      U     "MAL1S017Par".Ilo.GrCMDManStop[1];
      R     "MAL1S017Par".Ilo.GrCMDManStop[1];
// man fault reset
      U     "MAL1S017Par".Ilo.GrCMDManFaultReset[1];
      S     "G005G".Gr.CmdFaultReset; // GENERAL ELEMENTS GERM 1
      S     "G100M".Gr.CmdFaultReset; // Traveling  Drive Germatingbox 1
      S     "G104M".Gr.CmdFaultReset; // Turning Screws Germinationbox 1
      R     "MAL1S017Par".Ilo.GrCMDManFaultReset[1];
      NOP   0;
// Manual wall locking
      UN    "G099M".Gr.InManual; // Wall locking Germatingbox 1
      ON    "G102M".A_2115_KCL01I5.InpTrue; // pushbutton "locking"
      SPB   f102;
      S     "G099M".Gr.CmdOn; // Wall locking/unlocking Germatingbox 1
f102: NOP   0;
// Manual wall unlocking
      UN    "G099M".Gr.InManual; // Wall locking Germatingbox 1
      ON    "G102M".A_2115_KCL01I6.InpTrue; // pushbutton "unlocking"
      SPB   f103;
      S     "G099M".Gr.CmdOn; // Wall locking/unlocking Germatingbox 1
f103: NOP   0;
// Manual discharger coupling
      UN    "G098M".Gr.InManual; // discharger coupling Germatingbox 1
      ON    "G102M".A_2115_KCL01I4.InpTrue; // pushbutton "discharger coupling"
      SPB   f104;
      S     "G098M".Gr.CmdOn; // discharger coupling Germatingbox 1
f104: NOP   0;
// Manual discharger uncoupling
      UN    "G098M".Gr.InManual; // discharger coupling Germatingbox 1
      ON    "G102M".A_2115_KCL01I3.InpTrue; // pushbutton "discharger uncoupling"
      SPB   f105;
      S     "G098M".Gr.CmdOn; // discharger coupling Germatingbox 1
f105: NOP   0;
// Manual backwall moving
      UN    "G097M".Gr.InManual; // Backwall moving Germatingbox 1
      ON    "G102M".A_2115_KCL01I1.InpTrue; // pushbutton "backwall lifting"
      SPB   f106;
      S     "G097M".Gr.CmdOn; // Backwall moving Germatingbox 1
f106: NOP   0;
      UN    "G097M".Gr.InManual; // Backwall moving Germatingbox 1
      ON    "G102M".A_2115_KCL01I2.InpTrue; // pushbutton "backwall lowerring"
      SPB   f107;
      S     "G097M".Gr.CmdOn; // Backwall moving Germatingbox 1
f107: NOP   0;
// manual direction
      UN    "G100M".Gr.InManual; // Traveling  Drive Germatingbox 1
      O     ;
      UN    "G102M".A_2111_KCL01I3.InpTrue; // pushbutton "drive fwd"
      UN    "G102M".A_2111_KCL01I4.InpTrue; // pushbutton "drive rev"
      SPB   f109;
      U     "G102M".A_2111_KCL01I3.InpTrue; // pushbutton "drive fwd"
      =     "G100M".USW14; // ILO-cmd run fwd
      S     "G100M".Gr.CmdOn; // Traveling  Drive Germatingbox 1
      U     "G102M".A_2111_KCL01I4.InpTrue; // pushbutton "drive rev"
      =     "G100M".USW15; // ILO-cmd run rev
      S     "G100M".Gr.CmdOn; // Traveling  Drive Germatingbox 1

// target position
//      L     "MAL1S017Par".Ilo.SetpointInt01[1]
      L     20; // 20%
      T     "MAL1S017Par".Par.ParIntProcess.Speed_ILO_FloorRotating;
f109: NOP   0;

I10:  NOP   0;
//
// copy state
      U     "G100M".Gr.InOutAutostartMan; // TRAVELLING DRIVE GERM 1
      =     "MAL1S017Par".Ilo.GrSTMan[2];
      U     "G104M".Gr.InOutAutostartMan; // TURNING SCREWS GERM 1
      =     "MAL1S017Par".Ilo.GrSTMan[6];
      U     "G105M".Gr.InOutAutostartMan; // FAN AND VALVE SRAY AIR GERM 1
      =     "MAL1S017Par".Ilo.GrSTMan[7];
      U     "G106M".Gr.InOutAutostartMan; // FRESH AIR LOUVER GERM 1
      =     "MAL1S017Par".Ilo.GrSTMan[8];
      U     "G112M".Gr.InOutAutostartMan; // COOLING / HEATING GERM 1
      =     "MAL1S017Par".Ilo.GrSTMan[14];
NETWORK
TITLE =ASW_9999: Init ASW Flags
// clear all flags explicde to find them back
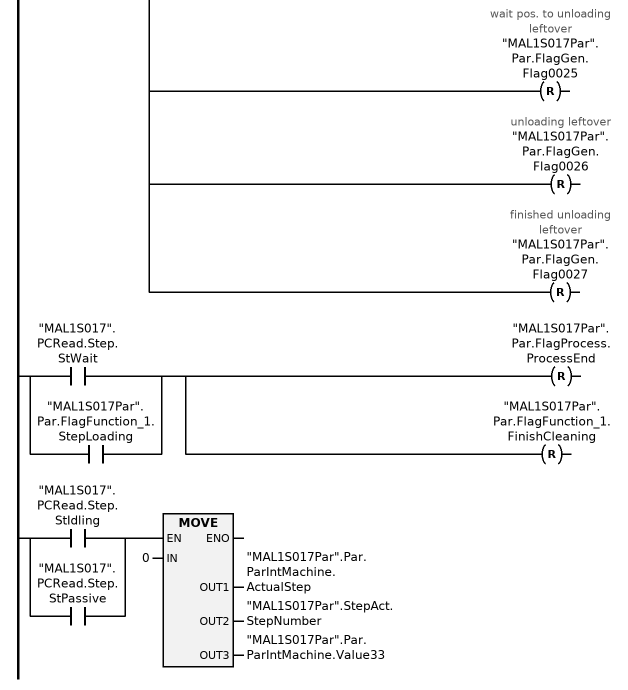
      U     "MAL1S017".PCRead.Step.StIdling;
      O     "MAL1S017".PCRead.Step.StPassive;
      R     "MAL1S017Par".Par.FlagFunction_1.StepLoading;
      R     "MAL1S017Par".Par.FlagFunction_1.StepUnloading;
      R     "MAL1S017Par".Par.FlagFunction_1.StepCleaning;
      R     "MAL1S017Par".Par.FlagFunction_1.LoadingBreak;
      R     "MAL1S017Par".Par.FlagFunction_1.UnloadingBreak;
      R     "MAL1S017Par".Par.FlagFunction_1.CleaningBreak;
      R     "MAL1S017Par".Par.FlagFunction_1.FinishLoading;
      R     "MAL1S017Par".Par.FlagFunction_1.FinishUnloading;
      R     "MAL1S017Par".Par.FlagFunction_1.FinishCleaning;
      R     "MAL1S017Par".Par.FlagFunction_1.Round_1;
      R     "MAL1S017Par".Par.FlagFunction_1.Round_2;
      R     "MAL1S017Par".Par.FlagFunction_1.Round_3;
      R     "MAL1S017Par".Par.FlagFunction_1.Round_4;
      R     "MAL1S017Par".Par.FlagFunction_1.Round_5;
      R     "MAL1S017Par".Par.FlagFunction_1.Round_6;
      R     "MAL1S017Par".Par.FlagFunction_1.Beladung_beendet;
      R     "MAL1S017Par".Par.FlagFunction_1.Entladerunden_erreicht;
      R     "MAL1S017Par".Par.FlagFunction_1.Reinigungsrunde_erreicht;
      R     "MAL1S017Par".Par.FlagGen.TurningStarted;
      R     "MAL1S017Par".Par.FlagFunction_1.TurningStart;
      R     "MAL1S017Par".Par.FlagFunction_1.TurningStop;
      R     "MAL1S017Par".Par.FlagFunction_1.TurningLeft;
      R     "MAL1S017Par".Par.FlagFunction_1.TurningRight;
      R     "MAL1S017Par".Par.FlagFunction_1.LoadFirstPartEnd;
      R     "MAL1S017Par".Par.FlagFunction_1.TurningWithSpraying;
      R     "MAL1S017Par".Par.FlagFunction_1.TurningWithoutSpraying;
      R     "MAL1S017Par".Par.FlagGen.TurningStarted;
      R     "MAL1S017Par".Par.FlagProcess2.Turning1WithoutSpraying;
      R     "MAL1S017Par".Par.FlagProcess2.Turning2WithoutSpraying;
      R     "MAL1S017Par".Par.FlagProcess2.Turning1WithSpraying;
      R     "MAL1S017Par".Par.FlagProcess2.Turning2WithSpraying;
      R     "MAL1S017Par".Par.FlagProcess2.Turning1WithDosing;
      R     "MAL1S017Par".Par.FlagProcess2.Turning2WithDosing;
      R     "MAL1S017Par".Par.FlagProcess2.StartFirstTurningRound;
      R     "MAL1S017Par".Par.FlagProcess2.StartSecondTurningRound;

      R     "MAL1S017Par".Par.FlagFunction_1.UnloadFirstPartEnd;
      R     "MAL1S017Par".Par.FlagFunction_1.UnloadSecondPartEnd;
      R     "MAL1S017Par".Par.FlagFunction_1.UnloadFirstPart;
      R     "MAL1S017Par".Par.FlagFunction_1.UnloadSecondPart;
      R     "MAL1S017Par".Par.FlagFunction_1.UnloadingStarted;
      R     "MAL1S017Par".Par.FlagProcess.ProcessActive;
      R     "MAL1S017Par".Par.FlagProcess.ProcessStartFP;
      R     "MAL1S017Par".Par.FlagProcess.ProcessStartScan;
      R     "MAL1S017Par".Par.FlagProcess.ProcessEnd;
      R     "MAL1S017Par".Par.FlagProcess.FP_SendResultToPIC;
      R     "MAL1S017Par".Par.FlagMachine.ImpulsNullstellung;
      R     "MAL1S017Par".Par.FlagMachine_0.CmdTurnRevAfterUnloading;
      R     "MAL1S017Par".Par.FlagMachine_0.CleaningAfterUnloading;
      R     "MAL1S017Par".Par.FlagMachine_0.CleaningAfterLoading;

      R     "MAL1S017Par".Par.FlagGen.Flag0024; // finished first unloading
      R     "MAL1S017Par".Par.FlagGen.Flag0025; // wait pos. to unloading leftover
      R     "MAL1S017Par".Par.FlagGen.Flag0026; // unloading leftover
      R     "MAL1S017Par".Par.FlagGen.Flag0027; // finished unloading leftover

//
      U     "MAL1S017".PCRead.Step.StWait;
      O     "MAL1S017Par".Par.FlagFunction_1.StepLoading;
      R     "MAL1S017Par".Par.FlagProcess.ProcessEnd;
      R     "MAL1S017Par".Par.FlagFunction_1.FinishCleaning;

      U     "MAL1S017".PCRead.Step.StIdling;
      O     "MAL1S017".PCRead.Step.StPassive;
      SPBN  csn;
      L     0; // clear step number
      T     "MAL1S017Par".Par.ParIntMachine.ActualStep;
      T     "MAL1S017Par".StepAct.StepNumber;
      T     "MAL1S017Par".Par.ParIntMachine.Value33; //aktuelle Wartezeit Maschine bei 100% Unloading-Position
csn:  NOP   0;
NETWORK
TITLE =Main0_End: Init flag
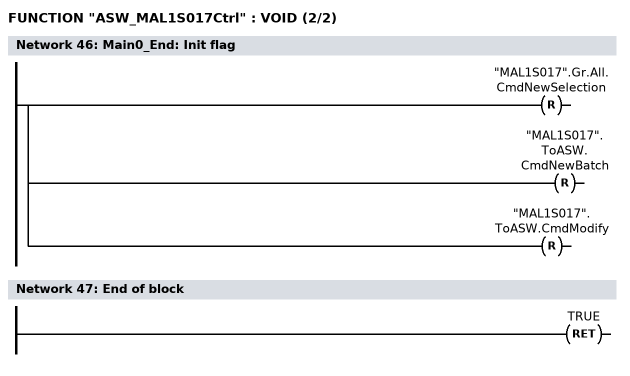

      SET   ;
      R     "MAL1S017".Gr.All.CmdNewSelection;
      R     "MAL1S017".ToASW.CmdNewBatch;
      R     "MAL1S017".ToASW.CmdModify;

NETWORK
TITLE =End of block

      BE    ;

END_FUNCTION

